// TIA Portal V17 export
// export: Created 2023-12-22T15:08:02.2560158Z, ExportSetting WithDefaults, DisplayName Totally Integrated Automation Portal, DisplayVersion V17, DisplayName TIA Portal Openness, DisplayVersion V17, DisplayName TIA Portal Version Control Interface, DisplayVersion V17, DisplayName STEP 7 Professional, DisplayVersion V17, DisplayName STEP 7 Safety, DisplayVersion V17, DisplayName WinCC Advanced, DisplayVersion V17
FUNCTION_BLOCK "DIx_1"   // FB200, LAD
{ S7_Optimized_Access := 'FALSE' }
VERSION : 0.1
// Input - входной сигнал контроллера
// pulse - частота фильтрации дребезга
// Signal - обработанный и отфильтрованный сигнал, используемый в дальнейшем
// stored: AutoNumber false, IsIECCheckEnabled false, SetENOAutomatically false, UDAEnableTagReadback false
   VAR
      AllBlock { S7_SetPoint := 'True'} : "DI_ex";   // Авар. блокировка / 2.4 разрешение на работу
      FS_Cl_1 { S7_SetPoint := 'True'} : "DI_ex";   // Датчик протока хлора 1 / 2.3 Нижний уровень
      FS_Cl_2 { S7_SetPoint := 'True'} : "DI_ex";   // Датчик протока хлора 2 / Ротаметр 1
      PS_PE { S7_SetPoint := 'True'} : "DI_ex";   // Питание датчиков камер давления / Ротаметр 2
      signal_5 { S7_SetPoint := 'True'} : "DI_ex";   // Ротаметр 3
      LS_KP_1_1 { S7_SetPoint := 'True'} : "DI_ex";   // Датчик затоплени КП1.1 LC5 / Датчик переливва
      LS_KP_1_2 { S7_SetPoint := 'True'} : "DI_ex";   // Датчик затоплени КП1.2 LC11 / Датчик переливва
      LS_KP_2_1 { S7_SetPoint := 'True'} : "DI_ex";   // Датчик затоплени КП2.1 LC6
      LS_KP_2_2 { S7_SetPoint := 'True'} : "DI_ex";   // Датчик затоплени КП2.2 LC16
      signal_10 { S7_SetPoint := 'True'} : "DI_ex";
      signal_11 { S7_SetPoint := 'True'} : "DI_ex";
      signal_12 { S7_SetPoint := 'True'} : "DI_ex";
   END_VAR
   VAR DB_SPECIFIC
      Time_DTL { S7_SetPoint := 'True'} : DTL;
   END_VAR
   VAR_TEMP   // added for the SCL form of the ladder/FBD networks
      _w1 : Bool;
      _w2 : Bool;
      _w3 : Bool;
   END_VAR
BEGIN

REGION Network 1: AllBlock
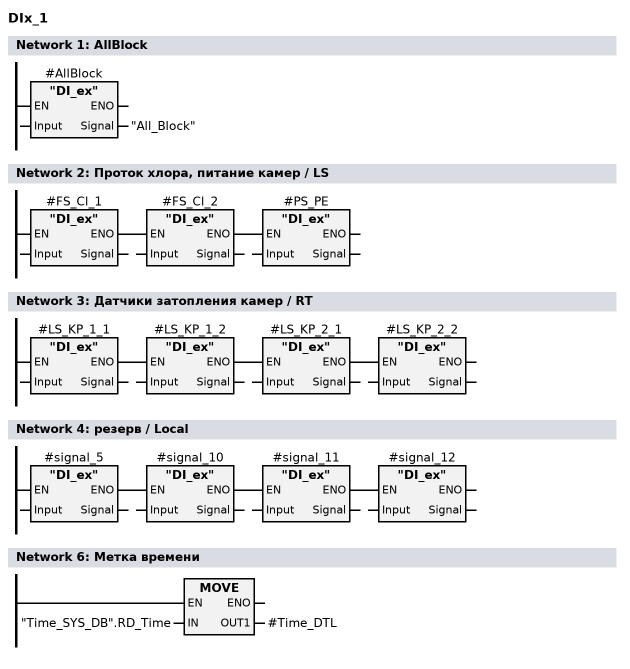
   RUNG wire#powerrail
      #AllBlock(Input :=, Signal => "All_Block")
   END_RUNG
   // the same network as SCL:
   #AllBlock(Signal => "All_Block");   // "DI_ex"
END_REGION

REGION Network 2: Проток хлора, питание камер / LS
   RUNG wire#powerrail
      #FS_Cl_1(Input :=, Signal =>)
      #FS_Cl_2(Input :=, Signal =>)
      #PS_PE(Input :=, Signal =>)
   END_RUNG
   // the same network as SCL:
   #FS_Cl_1(ENO => #_w1);   // "DI_ex"
   #FS_Cl_2(EN := #_w1, ENO => #_w2);   // "DI_ex"
   IF #_w2 THEN
       #PS_PE();   // "DI_ex"
   END_IF;
END_REGION

REGION Network 3: Датчики затопления камер / RT
   RUNG wire#powerrail
      #LS_KP_1_1(Input :=, Signal =>)
      #LS_KP_1_2(Input :=, Signal =>)
      #LS_KP_2_1(Input :=, Signal =>)
      #LS_KP_2_2(Input :=, Signal =>)
   END_RUNG
   // the same network as SCL:
   #LS_KP_1_1(ENO => #_w1);   // "DI_ex"
   #LS_KP_1_2(EN := #_w1, ENO => #_w2);   // "DI_ex"
   #LS_KP_2_1(EN := #_w2, ENO => #_w3);   // "DI_ex"
   IF #_w3 THEN
       #LS_KP_2_2();   // "DI_ex"
   END_IF;
END_REGION

REGION Network 4: резерв / Local
   RUNG wire#powerrail
      #signal_5(Input :=, Signal =>)
      #signal_10(Input :=, Signal =>)
      #signal_11(Input :=, Signal =>)
      #signal_12(Input :=, Signal =>)
   END_RUNG
   // the same network as SCL:
   #signal_5(ENO => #_w1);   // "DI_ex"
   #signal_10(EN := #_w1, ENO => #_w2);   // "DI_ex"
   #signal_11(EN := #_w2, ENO => #_w3);   // "DI_ex"
   IF #_w3 THEN
       #signal_12();   // "DI_ex"
   END_IF;
END_REGION

REGION Network 5: Авария
END_REGION

REGION Network 6: Метка времени
   RUNG wire#powerrail
      Move(in := "Time_SYS_DB".RD_Time, out1 => #Time_DTL)
   END_RUNG
   // the same network as SCL:
   #Time_DTL := "Time_SYS_DB".RD_Time;
END_REGION
END_FUNCTION_BLOCK
